// TIA Portal V20 export
TYPE "LER_typeUnitRecipe"
// stored: Access Published
   STRUCT
      processUnitNo : Int;
      selectedRecipeTypeID : Int;
      selectedRecipeID : Int;
      currentRecipeName : WString;
      currentRecipeID : Int;
      unitRecipe : "LER_typeRecipe";
   END_STRUCT;
END_TYPE
